TYPE Pucks :
STRUCT
	y 		 	: LREAL;
	zOffset		: LREAL;
	xOffset		: LREAL;
	code	 	: INT;
END_STRUCT
END_TYPE

(* stored: Version 1.1.0.1, ProductVersion 3.1.4024.11
   DUT Pucks: Id {7a92efe1-2e60-4fc2-aa81-c2fa8145568b} *)
